(* IEC 61131-3 sources: teller/JD_Teller_LC2_V11/Class/easyFileHandling, 1 file *)

(* ---- easyFileHandling.st ---- *)
(*!
<Class
	Name               = "easyFileHandling"
	Revision           = "0.0"
	RealtimeTask       = "false"
	CyclicTask         = "false"
	BackgroundTask     = "false"
	Sigmatek           = "false"
	OSInterface        = "false"
	HighPriority       = "false"
	Automatic          = "false"
	UpdateMode         = "Prescan"
	SharedCommandTable = "true"
	Objectsize         = "(660,600)">
	<Channels>
		<Server Name="ExtensionFilterStr" Class="String" Visualized="true" Initialize="true" WriteProtected="false" Retentive="false" Comment="use this channel to access the string functions"/>
		<Server Name="FileSelectedOK" Visualized="true" Initialize="false" WriteProtected="false" Retentive="false"/>
		<Server Name="FileStr" Class="String" Visualized="true" Initialize="true" WriteProtected="false" Retentive="false" Comment="use this channel to access the string functions"/>
		<Server Name="PathStr" Class="String" Visualized="true" Initialize="true" WriteProtected="false" Retentive="false" Comment="use this channel to access the string functions"/>
		<Server Name="toOpenFileSt" Class="String" Visualized="true" Initialize="true" WriteProtected="false" Retentive="false" Comment="use this channel to access the string functions"/>
		<Client Name="ExtensionFilter" Required="false" Internal="true"/>
		<Client Name="FileString" Required="false" Internal="true"/>
		<Client Name="PathString" Required="false" Internal="true"/>
		<Client Name="toOpenFileStr" Required="true" Internal="true"/>
	</Channels>
	<Network Name="easyFileHandling">
		<!-- List of Components in this network -->
		<Components>
			<Object
				Name       = "_base"
				Class      = "easyFileList"
				Position   = "(1201,120)"
				Visualized = "false">
				<Channels>
					<Server Name="DirectoryBack"/>
					<Server Name="Entries"/>
					<Server Name="Refresh"/>
					<Server Name="RefreshFiles"/>
					<Server Name="Server0"/>
					<Client Name="cToolCatLoadInfo"/>
					<Client Name="ExtensionFilter"/>
					<Client Name="FileIO"/>
					<Client Name="FileString"/>
					<Client Name="LineWidth" Value="0"/>
					<Client Name="Lse"/>
					<Client Name="PathString"/>
					<Client Name="toOpenFileString"/>
					<Client Name="VerticalLevel"/>
				</Channels>
			</Object>
			<Object
				Name       = "ExtensionFilter"
				Class      = "String"
				Position   = "(60,990)"
				Visualized = "true">
				<Channels>
					<Server Name="Data"/>
					<Client Name="SingleRealloc" Value="1"/>
				</Channels>
			</Object>
			<Object
				Name       = "FileString"
				Class      = "String"
				Position   = "(60,840)"
				Visualized = "true">
				<Channels>
					<Server Name="Data"/>
					<Client Name="SingleRealloc" Value="1"/>
				</Channels>
			</Object>
			<Object
				Name       = "PathString"
				Class      = "String"
				Position   = "(60,690)"
				Visualized = "true">
				<Channels>
					<Server Name="Data"/>
					<Client Name="SingleRealloc" Value="1"/>
				</Channels>
			</Object>
			<Object
				Name       = "toOpenFileStr"
				Class      = "String"
				Position   = "(60,1200)"
				Visualized = "true">
				<Channels>
					<Server Name="Data"/>
					<Client Name="SingleRealloc" Value="1"/>
				</Channels>
			</Object>
		</Components>
		<Comments>
		</Comments>
		<!-- List of Connections in this network -->
		<Connections>
			<Connection Source="_base.PathString" Destination="PathString.Data" Vertices="(1201,450),(780,450),(780,780),(376,780),"/>
			<Connection Source="this.Server0" Destination="_base.Server0" Vertices="(1673,210),(1501,210),"/>
			<Connection Source="this.Refresh" Destination="_base.Refresh" Vertices="(1673,270),(1501,270),"/>
			<Connection Source="_base.Lse" Destination="this.Lse" Vertices="(1201,210),(38,210),"/>
			<Connection Source="_base.FileString" Destination="FileString.Data" Vertices="(1201,510),(840,510),(840,930),(376,930),"/>
			<Connection Source="this.Entries" Destination="_base.Entries" Vertices="(1673,330),(1501,330),"/>
			<Connection Source="_base.FileIO" Destination="this.FileIO" Vertices="(1201,390),(1170,390),(1170,270),(38,270),"/>
			<Connection Source="this.PathStr" Destination="PathString.Data" Vertices="(1673,510),(1530,510),(1530,780),(376,780),"/>
			<Connection Source="this.FileStr" Destination="FileString.Data" Vertices="(1673,570),(1560,570),(1560,930),(660,930),(376,930),"/>
			<Connection Source="_base.ExtensionFilter" Destination="ExtensionFilter.Data" Vertices="(1201,570),(900,570),(900,1080),(376,1080),"/>
			<Connection Source="this.ExtensionFilterStr" Destination="ExtensionFilter.Data" Vertices="(1673,630),(1590,630),(1590,1080),(376,1080),"/>
			<Connection Source="this.toOpenFileStr" Destination="toOpenFileStr.Data"/>
			<Connection Source="_base.toOpenFileString" Destination="toOpenFileStr.Data" Vertices="(1201,630),(690,630),(690,1290),(376,1290),"/>
			<Connection Source="this.toOpenFileSt" Destination="toOpenFileStr.Data" Vertices="(1673,690),(1620,690),(1620,1290),(376,1290),"/>
			<Connection Source="this.DirectoryBack" Destination="_base.DirectoryBack" Vertices="(1673,390),(1501,390),"/>
			<Connection Source="this.RefreshFiles" Destination="_base.RefreshFiles" Vertices="(1673,450),(1501,450),"/>
			<Connection Source="_base.cToolCatLoadInfo" Destination="this.cToolCatLoadInfo" Vertices="(1201,690),(1140,690),(1140,330),(38,330),"/>
		</Connections>
		<!-- Headerfiles -->
		<Options>
		</Options>
	</Network>
</Class>
*)
#pragma using easyFileList

easyFileHandling : CLASS
: easyFileList
  //Servers:
	PathStr 	: SvrChCmd_UDINT;
	FileStr 	: SvrChCmd_UDINT;
	ExtensionFilterStr 	: SvrChCmd_UDINT;
	toOpenFileSt 	: SvrChCmd_UDINT;
	FileSelectedOK 	: SvrCh_UDINT;
  //Clients:
	virtual PathString 	: CltChCmd_String;
	virtual FileString 	: CltChCmd_String;
	virtual ExtensionFilter 	: CltChCmd_String;
	toOpenFileStr 	: CltChCmd_String;
  //Variables:
  //Functions:

	FUNCTION VIRTUAL GLOBAL Init;

	FUNCTION VIRTUAL GLOBAL ReadFiles;

	FUNCTION VIRTUAL GLOBAL PathStr::Read
		VAR_OUTPUT
			output (EAX) 	: UDINT;
		END_VAR;

	FUNCTION VIRTUAL GLOBAL PathStr::Write
		VAR_INPUT
			input (EAX) 	: UDINT;
		END_VAR
		VAR_OUTPUT
			result (EAX) 	: UDINT;
		END_VAR;

	FUNCTION VIRTUAL GLOBAL FileStr::Read
		VAR_OUTPUT
			output (EAX) 	: DINT;
		END_VAR;

	FUNCTION VIRTUAL GLOBAL FileStr::Write
		VAR_INPUT
			input (EAX) 	: UDINT;
		END_VAR
		VAR_OUTPUT
			result (EAX) 	: UDINT;
		END_VAR;

	FUNCTION VIRTUAL GLOBAL ExtensionFilterStr::Read
		VAR_OUTPUT
			output (EAX) 	: UDINT;
		END_VAR;

	FUNCTION VIRTUAL GLOBAL ExtensionFilterStr::Write
		VAR_INPUT
			input (EAX) 	: UDINT;
		END_VAR
		VAR_OUTPUT
			result (EAX) 	: UDINT;
		END_VAR;

	FUNCTION VIRTUAL GLOBAL toOpenFileSt::Read
		VAR_OUTPUT
			output (EAX) 	: DINT;
		END_VAR;

	FUNCTION VIRTUAL GLOBAL toOpenFileSt::Write
		VAR_INPUT
			input (EAX) 	: UDINT;
		END_VAR
		VAR_OUTPUT
			result (EAX) 	: UDINT;
		END_VAR;

	FUNCTION VIRTUAL GLOBAL FileSelectedOK::Read
		VAR_OUTPUT
			output (EAX) 	: UDINT;
		END_VAR;
  //Tables:
	FUNCTION @STD
		VAR_OUTPUT
			ret_code	: CONFSTATES;
		END_VAR;
	FUNCTION GLOBAL TAB @CT_;
END_CLASS;

#pragma using String

FUNCTION VIRTUAL GLOBAL easyFileHandling::PathStr::Read
	VAR_OUTPUT
		output (EAX) 	: UDINT;
	END_VAR

	PathStr := PathString.Data.Read();
	output := PathStr;

END_FUNCTION

FUNCTION VIRTUAL GLOBAL easyFileHandling::PathStr::Write
	VAR_INPUT
		input (EAX) 	: UDINT;
	END_VAR
	VAR_OUTPUT
		result (EAX) 	: UDINT;
	END_VAR

	PathStr := input;
 	result := PathString.Data.Write(PathStr);

END_FUNCTION

FUNCTION VIRTUAL GLOBAL easyFileHandling::FileStr::Read
	VAR_OUTPUT
		output (EAX) 	: DINT;
	END_VAR

	FileStr := FileString.Data.Read();
	output := FileStr$DINT;

END_FUNCTION

FUNCTION VIRTUAL GLOBAL easyFileHandling::FileStr::Write
	VAR_INPUT
		input (EAX) 	: UDINT;
	END_VAR
	VAR_OUTPUT
		result (EAX) 	: UDINT;
	END_VAR

	FileStr := input;
 	result := FileString.Data.Write(FileStr);

END_FUNCTION

FUNCTION VIRTUAL GLOBAL easyFileHandling::ExtensionFilterStr::Read
	VAR_OUTPUT
		output (EAX) 	: UDINT;
	END_VAR

	ExtensionFilterStr := ExtensionFilter.Data.Read();
	output := ExtensionFilterStr$UDINT;

END_FUNCTION

FUNCTION VIRTUAL GLOBAL easyFileHandling::ExtensionFilterStr::Write
	VAR_INPUT
		input (EAX) 	: UDINT;
	END_VAR
	VAR_OUTPUT
		result (EAX) 	: UDINT;
	END_VAR

	ExtensionFilterStr$UDINT := input;
 	result := ExtensionFilter.Data.Write(ExtensionFilterStr);

END_FUNCTION

FUNCTION VIRTUAL GLOBAL easyFileHandling::toOpenFileSt::Read
	VAR_OUTPUT
		output (EAX) 	: DINT;
	END_VAR

	toOpenFileSt := toOpenFileStr.Data.Read();
	output := toOpenFileSt$DINT;

END_FUNCTION

FUNCTION VIRTUAL GLOBAL easyFileHandling::toOpenFileSt::Write
	VAR_INPUT
		input (EAX) 	: UDINT;
	END_VAR
	VAR_OUTPUT
		result (EAX) 	: UDINT;
	END_VAR

	toOpenFileSt := input;
 	result := toOpenFileStr.Data.Write(toOpenFileSt);

END_FUNCTION

FUNCTION VIRTUAL GLOBAL easyFileHandling::Init

  StartPathLen := PathString.GetLength();
  PathString.ReadDataOff(udOff:=0, pData:=#StartPath[0], udMax:=StartPathLen);
  StartPath[StartPathLen] :=0;

END_FUNCTION

FUNCTION VIRTUAL GLOBAL easyFileHandling::ReadFiles
  easyFileList::ReadFiles();
  InsertCmd(Cmd_Redraw, 0, 0);
END_FUNCTION

FUNCTION VIRTUAL GLOBAL easyFileHandling::FileSelectedOK::Read
	VAR_OUTPUT
		output (EAX) 	: UDINT;
	END_VAR

//  FileSelectedOK := toOpenFileStr.GetLength()>1;

//	if toOpenFileStr.GetLength()>1 then
//    FileSelectedOK:=1;
//  else
//    FileSelectedOK:=0;
//  end_if;

FileSelectedOK := toOpenFileStr.GetLength();

	output := FileSelectedOK;

END_FUNCTION
